// TwinCAT 3 PLC project PRG_B_HMIManager
// Title: B_HMIManager
// Company: RafałOS
// Author: Rafał Osajda
// ProjectVersion: 0.0.0.7
// ProgramVersion: 3.1.4024.0
// libraries:
//   B_Base, * (RafalOS)
//   B_Base_HMI_Connector, * (RafalOS)
//   B_HMIElements, * (RafalOS)
//   B_MachineControl, * (RafalOS)
//   B_MachineControl_HMI_Connector, * (RafalOS)
//   B_StatesAndModes, * (RafalOS)
//   Tc2_Standard, * (Beckhoff Automation GmbH)
//   Tc2_System, * (Beckhoff Automation GmbH)
//   Tc3_Module, * (Beckhoff Automation GmbH)
// project tree:
//   / PlcTask.TcTTO (not stored)
//   POUs Compilation/ PRG_Compilation.TcPOU
//   POUs/01_HMIManager/ FB_HMIManager.TcPOU, ITF_HMIManager.TcIO, ITF_HMIManagerConfigure.TcIO, ST_HMIManager.TcDUT
//   POUs/02_Configuration/ FB_HMIConfigure.TcPOU, ITF_HMIConfiguration.TcIO, ITF_HMIConfigure.TcIO

// ---- POUs/01_HMIManager/ST_HMIManager.TcDUT
TYPE ST_HMIManager EXTENDS ST_BaseGroupElement_HMI_Link :
STRUCT
	stMainMenu			: ST_HMIEMenu_HMI_Link;
	
END_STRUCT
END_TYPE

// ---- POUs/01_HMIManager/ITF_HMIManager.TcIO
INTERFACE ITF_HMIManager EXTENDS ITF_BaseGroupElement

END_INTERFACE

// ---- POUs/01_HMIManager/ITF_HMIManagerConfigure.TcIO
INTERFACE ITF_HMIManagerConfigure EXTENDS ITF_Base

(*			
	RafalOS
	Rafał Osajda		19.11.2025		TC 4024.66
	Dodanie połączenia do MachineControl  wywoływane z konfiguracji
*)
METHOD AddMachineControlConnectorFromConfiguration : BOOL
VAR_INPUT
	itfMachineControl	: ITF_MachineControl_HMI;
END_VAR
END_METHOD

(*			
	RafalOS
	Rafał Osajda		14.11.2025		TC 4024.66
	Dodanie do systemu menu głównego 
*)
METHOD PUBLIC AddMainMenuFromConfiguration : BOOL
VAR_INPUT
	fbMenu			: ITF_HMIEMenu;
	fbMenu_HMI		: ITF_HMIEMenu_HMI;
END_VAR
END_METHOD

METHOD PUBLIC GetNumberOfAddedButtons : INT
VAR_INPUT
END_VAR
END_METHOD

(*			
	RafalOS
	Rafał Osajda		18.11.2025		TC 4024.66
	Podłączenie głównej struktury danych dla domyślnych elementów 
*)
METHOD LinkHMIManagerDataFromConfiguration : BOOL
VAR_INPUT
	stData					: REFERENCE TO ST_HMIManager;
END_VAR
END_METHOD

(*			
	RafalOS
	Rafał Osajda		18.11.2025		TC 4024.66
	Ustawia przycisk na aktywny  - pierwsze okno w wyświetlaniu wizualizacji - wywoływane z konfiguracji
*)
METHOD SetButtonActiveFromConfiguration : BOOL
VAR_INPUT
	iNumber		: INT;	//numr przycisku
	bValue		: BOOL;
END_VAR
END_METHOD

(*			
	RafalOS
	Rafał Osajda		18.11.2025		TC 4024.66
	Ustawia przyciski na wlaczone lub wylaczone - możliwośc naciśnięcia
*)
METHOD SetButtonsEnabledFromConfiguration : BOOL
VAR_INPUT
	iNumber		: INT;	//numr przycisku
	bValue		: BOOL;
END_VAR
END_METHOD

(*			
	RafalOS
	Rafał Osajda		18.11.2025		TC 4024.66
	Ustawia przyciski na widoczne lub nie widoczne
*)
METHOD SetButtonsVisibleFromConfiguration : BOOL
VAR_INPUT
	iNumber		: INT;	//numr przycisku
	bValue		: BOOL;
END_VAR
END_METHOD

END_INTERFACE

// ---- POUs/02_Configuration/ITF_HMIConfiguration.TcIO
INTERFACE ITF_HMIConfiguration

(*			
	RafalOS
	Rafał Osajda		19.11.2025		TC 4024.66
	Dodanie połączenia do MachineControl
*)
METHOD AddMachineControlConnector : BOOL
VAR_INPUT
	itfHMIManager	: ITF_HMIManagerConfigure;
END_VAR
END_METHOD

(*			
	RafalOS
	Rafał Osajda		14.11.2025		TC 4024.66
	Dodanie do systemu menu głównego 
*)
METHOD PUBLIC AddMainMenu : BOOL
VAR_INPUT
	itfHMIManager	: ITF_HMIManagerConfigure;
END_VAR
END_METHOD

(*			
	RafalOS
	Rafał Osajda		19.11.2025		TC 4024.66
	Dodanie modułów do przygotowywania stron do wyświetlenia
*)
METHOD AddPrepareScreenModule : BOOL
VAR_INPUT
	itfHMIManager	: ITF_HMIManagerConfigure;
END_VAR
END_METHOD

(*			
	RafalOS
	Rafał Osajda		18.11.2025		TC 4024.66
	Podłączenie głównej struktury danych dla domyślnych elementów 
*)
METHOD LinkHMIManagerData : BOOL
VAR_INPUT
	itfHMIManager	: ITF_HMIManagerConfigure;
END_VAR
END_METHOD

(*			
	RafalOS
	Rafał Osajda		18.11.2025		TC 4024.66
	Ustawia przycisk na aktywny  - pierwsze okno w wyświetlaniu wizualizacji
*)
METHOD SetButtonActive : BOOL
VAR_INPUT
	itfHMIManager	: ITF_HMIManagerConfigure;
END_VAR
END_METHOD

(*			
	RafalOS
	Rafał Osajda		18.11.2025		TC 4024.66
	Ustawia przyciski na wlaczone lub wylaczone - możliwośc naciśnięcia
*)
METHOD SetButtonsEnabled : BOOL
VAR_INPUT
	itfHMIManager	: ITF_HMIManagerConfigure;
END_VAR
END_METHOD

(*			
	RafalOS
	Rafał Osajda		18.11.2025		TC 4024.66
	Ustawia przyciski na widoczne lub nie widoczne
*)
METHOD SetButtonsVisible : BOOL
VAR_INPUT
	itfHMIManager	: ITF_HMIManagerConfigure;
END_VAR
END_METHOD

END_INTERFACE

// ---- POUs/02_Configuration/ITF_HMIConfigure.TcIO
INTERFACE ITF_HMIConfigure

METHOD PUBLIC AddConfiguration : BOOL
VAR_INPUT
	fbConfigure		: ITF_HMIConfiguration;
END_VAR
END_METHOD

METHOD PUBLIC Configure : BOOL
VAR_INPUT
	fbHMIManager			: ITF_HMIManagerConfigure;
END_VAR
END_METHOD

END_INTERFACE

// ---- POUs Compilation/PRG_Compilation.TcPOU
PROGRAM PRG_Compilation
VAR
	fbHMIManager		: FB_HMIManager;
	fbHMIConfigure		: FB_HMIConfigure;
	
END_VAR

END_PROGRAM

// ---- POUs/01_HMIManager/FB_HMIManager.TcPOU
FUNCTION_BLOCK FB_HMIManager EXTENDS FB_BaseGroupElement IMPLEMENTS ITF_HMIManager, ITF_HMIManagerConfigure
VAR
	(*	Inicjalizacja		*)
	bInitializeCycle			: BOOL;
	bInitDone					: BOOL;
	bIsValidData				: bool;
	(*	Konfiguracja		*)
	itfHMIConfigure				: ITF_HMIConfigure;		//moduł konfiguracji
	(*	Menu główne	*)
	itfMainMenu					: ITF_HMIEMenu;
	itfMainMenuHMI				: ITF_HMIEMenu_HMI;
	iNumberOfButtonMainMenu		: INT;
	iNumberOfActiveScreen		: INT;
	iNumberOfPreviewScreen		: INT;
	bChangePage					: BOOL;
	(*	Obsługa zmiany strony	*)
	arrChangePageSupport		: ARRAY [0..GVL_HMIEConstans.MAX_NUMBER_OF_BUTTON_IN_MENU] OF 
									ARRAY [0..GVL_SaMConstans.NUMBER_OF_MODES] OF ITF_ChangePageSupport;
	(*	Dana wspólne dla całego systemu	*)
	refstManagerData			: REFERENCE TO ST_HMIManager;
END_VAR

IF (NOT THIS^.bInitializeCycle) THEN
	THIS^.bInitializeCycle		:= TRUE;
	THIS^.bInitDone				:= THIS^.InitializeCycle ();
ELSIF (THIS^.bInitDone) THEN
	THIS^.ExecuteCycle ();
END_IF

(*			
	RafalOS
	Rafał Osajda		14.11.2025		TC 4024.66
	Dodanie do systemu menu głównego 
*)
METHOD PUBLIC AddMainMenuFromConfiguration : BOOL
VAR_INPUT
	fbMenu			: ITF_HMIEMenu;
	fbMenu_HMI		: ITF_HMIEMenu_HMI;
END_VAR
THIS^.SetText (eLocation := E_BaseLocation.pl, wsDescription := "Menu główne");
THIS^.SetText (eLocation := E_BaseLocation.en, wsDescription := "Main menu");
THIS^.SetText (eLocation := E_BaseLocation.de, wsDescription := "Hauptmenü");
fbMenu.SetName (stName := THIS^.GetTexts ());
THIS^.AddControlElement (itfControlElement := fbMenu);

THIS^.itfMainMenu := fbMenu;
THIS^.itfMainMenu.LinkCommonData (stCommonData := THIS^.refstCommonData);

THIS^.itfMainMenuHMI  := fbMenu_HMI;
THIS^.itfMainMenuHMI.LinkCommonData (stCommonData := THIS^.refstCommonData);
END_METHOD

(*			
	RafalOS
	Rafał Osajda		29.10.2025		TC 4024.66
	Dodawanie intefejsu konfiguracji
*)
METHOD PUBLIC AddModulConfigure : BOOL
VAR_INPUT
	fbHMIConfigure			: ITF_HMIConfigure;
END_VAR
THIS^.itfHMIConfigure		:= fbHMIConfigure;
END_METHOD

(*			
	RafalOS
	Rafał Osajda		10.11.2025		TC 4024.66
	Główna metoda sterujaca wyświetlaniem dsanych na HMI
*)
METHOD PUBLIC ExecuteCycle
	(* Testowanie MenuGlownego	*)
THIS^.itfMainMenu.Testing ();
	(*	Przepisanie Aktualnych zmiennych menu do struktury danych HMI	*)

THIS^.itfMainMenuHMI.PrepareDataForHMI ();
	
	(*	Aktualizacja zmiennych przy zmianie strony	*)
THIS^.bChangePage := THIS^.itfMainMenuHMI.IsChangePage ();

IF (THIS^.bChangePage) THEN
	THIS^.itfMainMenu.ResetChangePage ();
	THIS^.iNumberOfPreviewScreen := THIS^.itfMainMenuHMI.GetNumberOfPreviewScreen ();
	THIS^.iNumberOfActiveScreen := THIS^.itfMainMenuHMI.GetNumberOfActiveScreen ();

//	IF (THIS^.arrChangePageSupport [THIS^.iNumberOfPreviewScreen] <> 0) THEN
//		THIS^.arrChangePageSupport [THIS^.iNumberOfPreviewScreen].ClaerAfterPage ();
//	END_IF
//	IF (THIS^.arrChangePageSupport [THIS^.iNumberOfActiveScreen] <> 0) THEN
//		THIS^.arrChangePageSupport [THIS^.iNumberOfActiveScreen].PreparePage ();
//	END_IF
END_IF

	(*	Odświerzenia strrony 	*)
//IF (THIS^.arrChangePageSupport [THIS^.iNumberOfActiveScreen] <> 0) THEN
//	THIS^.arrChangePageSupport [THIS^.iNumberOfActiveScreen].PrepareDataForHMI ();
	//wyczyszczenie po ramce 
	//przygotowanie ramki
//END_IF
	(*	Skasowanie flagi zmiany strony	*)
END_METHOD

METHOD FB_init : BOOL
VAR_INPUT
	bInitRetains : BOOL; // if TRUE, the retain variables are initialized (warm start / cold start)
	bInCopyCode : BOOL;  // if TRUE, the instance afterwards gets moved into the copy code (online change)
END_VAR
THIS^.SetText (eLocation := E_BaseLocation.pl, wsDescription := "HMI Menadżer");
THIS^.SetText (eLocation := E_BaseLocation.en, wsDescription := "HMI Manager");
THIS^.SetText (eLocation := E_BaseLocation.de, wsDescription := "HMI Manager");
THIS^.SetName (stName := THIS^.GetTexts ());
END_METHOD

METHOD PUBLIC GetNumberOfAddedButtons : INT
VAR_INPUT
END_VAR
GetNumberOfAddedButtons := THIS^.itfMainMenu.GetNumberOfAddedButton ();
END_METHOD

METHOD PRIVATE InitializeCycle : BOOL
VAR
	bResult					: BOOL;
	iI: INT;
END_VAR
bResult				:= TRUE;

bResult				:= bResult AND THIS^.itfHMIConfigure.Configure (fbHMIManager := THIS^);

InitializeCycle		:= bResult;
END_METHOD

(*			
	RafalOS
	Rafał Osajda		18.11.2025		TC 4024.66
	Podłączenie głównej struktury danych dla domyślnych elementów 
*)
METHOD LinkCommonStructureDataFromConfiguration : BOOL
VAR_INPUT
	stData			: reference to ST_HMIManager;
END_VAR
THIS^.refstManagerData REF= stData;
END_METHOD

METHOD LinkHMIManagerDataFromConfiguration : BOOL
VAR_INPUT
	stData					: REFERENCE TO ST_HMIManager;
END_VAR
THIS^.refstManagerData	REF= stData;

THIS^.itfMainMenuHMI.LinkHMIEMenuData (stData := stData.stMainMenu);



IF (__ISVALIDREF (THIS^.refstManagerData)) THEN
	THIS^.bIsValidData := TRUE;
	LinkHMIManagerDataFromConfiguration := TRUE;
END_IF
END_METHOD

(*			
	RafalOS
	Rafał Osajda		18.11.2025		TC 4024.66
	Ustawia przycisk na aktywny  - pierwsze okno w wyświetlaniu wizualizacji - wywoływane z konfiguracji
*)
METHOD SetButtonActiveFromConfiguration : BOOL
VAR_INPUT
	iNumber		: INT;	//numr przycisku
	bValue		: BOOL;
END_VAR
THIS^.itfMainMenu.SetActiveButton (iButton := iNumber, bIN := bValue);
END_METHOD

(*			
	RafalOS
	Rafał Osajda		18.11.2025		TC 4024.66
	Ustawia przyciski na wlaczone lub wylaczone - możliwośc naciśnięcia
*)
METHOD SetButtonsEnabledFromConfiguration : BOOL
VAR_INPUT
	iNumber		: INT;	//numr przycisku
	bValue		: BOOL;
END_VAR
THIS^.itfMainMenu.SetEnableButton (iButton := iNumber, bIN := bValue);
END_METHOD

(*			
	RafalOS
	Rafał Osajda		18.11.2025		TC 4024.66
	Ustawia przyciski na widoczne lub nie widoczne
*)
METHOD SetButtonsVisibleFromConfiguration : BOOL
VAR_INPUT
	iNumber		: INT;	//numr przycisku
	bValue		: BOOL;
END_VAR
THIS^.itfMainMenu.SetVisibleButton (iButton := iNumber, bIN := bValue);
END_METHOD

END_FUNCTION_BLOCK

// ---- POUs/02_Configuration/FB_HMIConfigure.TcPOU
FUNCTION_BLOCK FB_HMIConfigure EXTENDS FB_Base IMPLEMENTS ITF_HMIConfigure
VAR
	(*	Baza konfiguracji	*)
	arritfConfigure				: ARRAY [1..10] OF ITF_HMIConfiguration;
	iNubmerOfAddedConfigure		: INT;
END_VAR

METHOD PUBLIC AddConfiguration : BOOL
VAR_INPUT
	fbConfigure		: ITF_HMIConfiguration;
END_VAR
IF (THIS^.iNubmerOfAddedConfigure + 1 <= 10) THEN
	THIS^.iNubmerOfAddedConfigure	:= THIS^.iNubmerOfAddedConfigure + 1;
	THIS^.arritfConfigure [THIS^.iNubmerOfAddedConfigure]	:= fbConfigure;
	AddConfiguration	:= TRUE;
ELSE
	AddConfiguration	:= FALSE;
END_IF
END_METHOD

METHOD PUBLIC Configure : BOOL
VAR_INPUT
	fbHMIManager			: ITF_HMIManagerConfigure;
END_VAR
VAR
	bResult				: BOOL;
	iI					: INT;
END_VAR
bResult			:= TRUE;

THIS^.arritfConfigure [1].AddMainMenu (itfHMIManager := fbHMIManager);
THIS^.arritfConfigure [1].LinkCommonStructureData (itfHMIManager := fbHMIManager);

FOR iI := 1 TO THIS^.iNubmerOfAddedConfigure DO 
	IF (THIS^.arritfConfigure [iI] <> 0) THEN
		THIS^.arritfConfigure [iI].SetButtonActive (itfHMIManager	:= fbHMIManager);
		THIS^.arritfConfigure [iI].SetButtonsVisible (itfHMIManager	:= fbHMIManager);
		THIS^.arritfConfigure [iI].SetButtonsEnabled (itfHMIManager	:= fbHMIManager);
		//THIS^.arritfConfigure [iI].

	END_IF
END_FOR

THIS^.arritfConfigure [1].LinkHMIManagerData (itfHMIManager := fbHMIManager);

Configure		:= bResult;
END_METHOD

END_FUNCTION_BLOCK
